TYPE ST_SetHW_Inputs :
(**************************************************************************************
 * 	Application		:	BoxControl Framework
 *	Revision		:	$Revision: 404529 $
 *	Revision date	:	$Date: 2018-04-23 08:21:38 +0200 (Mo., 23 Apr 2018) $
 *	Last changed by	:	$Author: b7bolm $
 *	URL				:	$URL: http://almscdc.swisslog.com/repo/SWPD/Development/BoxControlFramework/20_Release/trunk/01_Software/BCF/BCF/JumpStart/20_Product/11_Emu/12_E_Functions/10_Lib/10_Conv/10_Functions/01_DUTs/ST_SetHW_Inputs.TcDUT $
 *
 *	Purpose			:	Product type registration access - Conveyor
 *
 * ------------------------------------------------------------------------------------
 *	Copyright Swisslog [IP AG], Switzerland. All rights reserved.
 * 
 * ------------------------------------------------------------------------------------
 *	
 * 	Revision History: 
 *
 * 	VERSION			DATE			INITIALS			DESCRIPTION
 *	0.1				01.01.2001		swl					Example
 *
 **************************************************************************************)
STRUCT
	Occupied 		: ARRAY [1..9] OF BOOL; // Occupied sensor
	DriveRunning 	: ARRAY [1..9] OF BOOL; // Feedback signal drive is running
	HW_Input		: ARRAY [1..10] OF BOOL; // None specific HW inputs
END_STRUCT
END_TYPE

(* stored: Version 1.1.0.1, ProductVersion 3.1.4022.12
   DUT ST_SetHW_Inputs: Id {cacb7d81-7890-4700-8abd-0d8f44b621f9} *)
